Staubli VAL3: Tester.dtx

mdesc mNomSpeed
tool tTool = {z=110, fatherId=flange[0], ioLink=valve1}
public sio sSioOrdenador = {link=Socket\Feedback}
num l_nNumero
string sMessage
jointRx JHome = {j3=0.600000023841858}
jointRx JApproach1 = {j1=-7.51951662048618, j2=-3.64591570536508, j3=61.4224158850639, j4=1.01386296296635E-05, j5=122.22350312171, j6=172.480485827149}
pointRx PGet = {x=336.755109049414, y=-333.263434847665, z=-17.5292162192054, rx=-179.003488571719, ry=2.52863969251374E-06, rz=8.41296103690271E-07, fatherId=world[0]}
num nTest
